(* LS Electric XG5000 project: HMI *)
(* PLC LSPLC *)

PROGRAM NewProgram (* task: 스캔 프로그램 *)
VAR
    INST : TP;
    INST1 : TP;
    INST2 : TP;
END_VAR

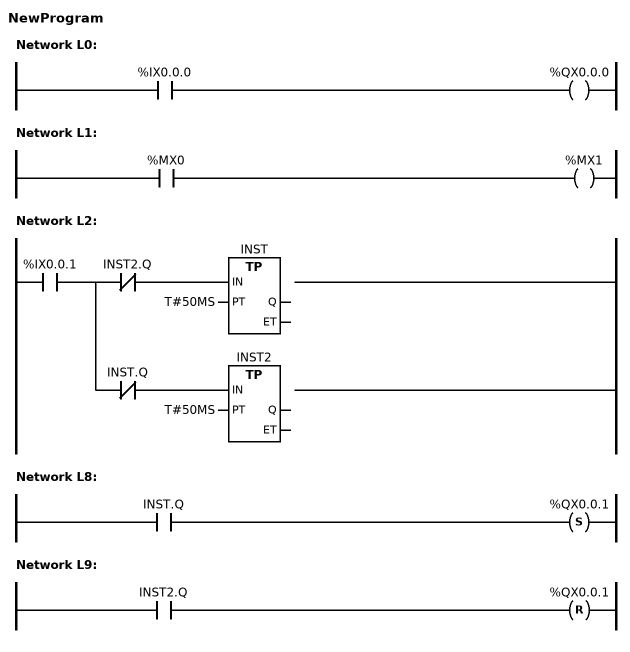
(* Rung L0 *)
%QX0.0.0 := %IX0.0.0;
(* Rung L1 *)
%MX1 := %MX0;
(* Rung L2 *)
INST(IN := %IX0.0.1 AND NOT INST2.Q, PT := T#50MS);
INST2(IN := %IX0.0.1 AND NOT INST.Q, PT := T#50MS);
(* Rung L8 *)
IF INST.Q THEN %QX0.0.1 := TRUE; END_IF;
(* Rung L9 *)
IF INST2.Q THEN %QX0.0.1 := FALSE; END_IF;
END_PROGRAM